PROGRAM cip
VAR
	ed_routine_starting_idle: BOOL;
	idle_redox_doser_enable: BOOL;
	
	tmr_idle_pumps: TON;
	idle_u_3112_b_request: BOOL;
	idle_u_3312_b_request: BOOL;
	idle_u_3405_b_request: BOOL;
	idle_u_3212_b_request: BOOL;
	tmr_idle_pump_delay: TON;
	u_3112_b_running: BOOL;
	u_3112_b_speed_ref: INT;
	u_3112_b_sp: REAL;
	salt_pressure_actual: REAL;
	idle_u_3112_b_ready: BOOL;
	u_3212_b_running: BOOL;
	idle_u_3212_b_ready: BOOL;
	idle_u_3312_b_ready: BOOL;
	u_3312_b_running: BOOL;
	u_3405_b_running: BOOL;
	idle_u_3405_b_ready: BOOL;
	idle_stack_power_enable: BOOL;
	ed_routine_cip: BOOL;
	
		nv_3110_b_open_request: BOOL;
	nv_3210_b_open_request: BOOL;
	nv_3310_b_open_request: BOOL;
	nv_3110_b_open_feedback: BOOL;
	nv_3210_b_open_feedback: BOOL;
	nv_3310_b_open_feedback: BOOL;
	cip_redox_doser_enable: BOOL;
	nv_3372_b_open_request: BOOL;
	nv_3135_b_open_request: BOOL;
	nv_3235_b_open_request: BOOL;
	nv_3335_b_open_request: BOOL;
	nv_3372_b_open_feedback: BOOL;
	nv_3135_b_open_feedback: BOOL;
	nv_3235_b_open_feedback: BOOL;
	nv_3335_b_open_feedback: BOOL;
	tmr_cip_pump_delay: TON;
	idle_u_3370_b_request: BOOL;
	u_3370_b_running: BOOL;
	u_3370_b_sp: REAL;
	tmr_cip_pump_start_delay: TON;
	tmr_cip_run: TON;
	cip_tmr_preset: TIME;
	
	u_3370_b_actual: INT; // What would this be???
	ft_3122_b_tot: INT;
	ft_3222_b_tot: INT;
	ft_3322_b_tot: INT;
	cip_flush_tot: INT;
	cip_flush_sp: INT;
	cip_u_3370_b_request: BOOL;
	cip_complete: BOOL;
	cip_stop_request: BOOL;
	nv_3372_b_cip_request: BOOL;
	nv_3135_b_cip_request: BOOL;
	nv_3235_b_cip_request: BOOL;
	nv_3335_b_cip_request: BOOL;
	redox_doser_cip_enable: BOOL;
	u_3370_b_cip_request: BOOL;
	CIP_TEMP_BIT: BOOL;
	tmr_cip_valve_delay: TON;
	tmr_cip_valve_delay_pt: TIME:= T#30S;
	tmr_cip_valve_delay_et: TIME;
	tmr_cip_valve_delay_q: BOOL;
	u_3112_b_cip_pressure_setpoint_request: REAL;
	u_3370_b_cip_pressure_setpoint_request: REAL;
END_VAR
VAR // added by the converter: edge detectors and wires of the graphical bodies
    _w1, _w2, _w3 : BOOL;
END_VAR

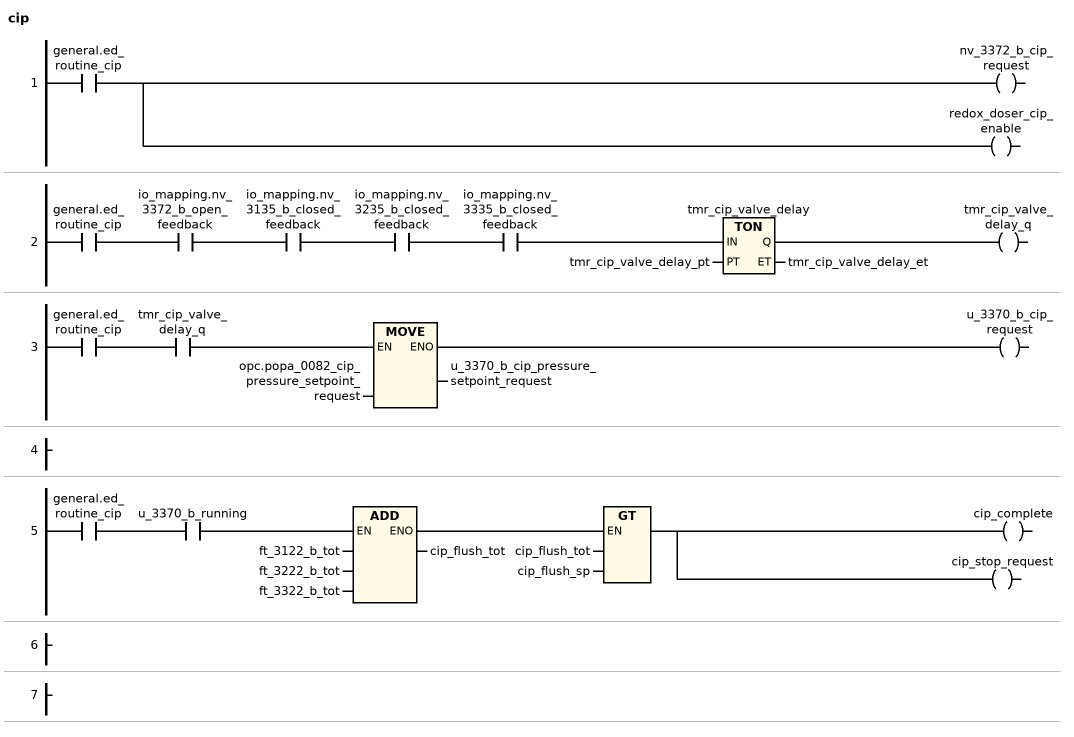
// NETWORK 1
nv_3372_b_cip_request := general.ed_routine_cip;
redox_doser_cip_enable := general.ed_routine_cip;

// NETWORK 2
tmr_cip_valve_delay(
    IN := general.ed_routine_cip AND io_mapping.nv_3372_b_open_feedback AND io_mapping.nv_3135_b_closed_feedback AND io_mapping.nv_3235_b_closed_feedback AND io_mapping.nv_3335_b_closed_feedback,
    PT := tmr_cip_valve_delay_pt,
    ET => tmr_cip_valve_delay_et); // TON
tmr_cip_valve_delay_q := tmr_cip_valve_delay.Q;

// NETWORK 3
_w1 := general.ed_routine_cip AND tmr_cip_valve_delay_q;
IF _w1 THEN u_3370_b_cip_pressure_setpoint_request := opc.popa_0082_cip_pressure_setpoint_request; END_IF
u_3370_b_cip_request := _w1;

// NETWORK 4

// NETWORK 5
_w2 := general.ed_routine_cip AND u_3370_b_running;
IF _w2 THEN cip_flush_tot := ft_3122_b_tot + ft_3222_b_tot + ft_3322_b_tot; END_IF
_w3 := _w2 AND cip_flush_tot > cip_flush_sp;
cip_complete := _w3;
cip_stop_request := _w3;

// NETWORK 6

// NETWORK 7

END_PROGRAM

(* stored: Version 1.1.0.1, ProductVersion 3.1.4024.15
   POU cip: Id {229a4917-364b-4aed-993d-1b6b88976092}, SpecialFunc None *)
